{attribute 'qualified_only'}
{attribute 'strict'}
{attribute 'to_string'}
TYPE E_EventType :
(
	Alarm := 0,
	Message := 1
);
END_TYPE

(* stored: Version 1.1.0.1
   DUT E_EventType: Id {d33035b2-8869-4a26-94a8-c90dc13e2fab} *)
